PROGRAM MAIN
VAR
	onTimer, offTimer : ton;
	
	start : BOOL;
END_VAR

onTimer(PT:=T#1S, Q=> GVL.imAlive);
offTimer(IN:= GVl.imAlive, PT:=T#1S);
IF offTimer.Q THEN
	onTimer.IN := FALSE;
END_IF
IF NOT GVL.imAlive AND NOT onTimer.IN THEN
	onTimer.IN := TRUE;
	GVL.counter := GVL.counter +1;
END_IF

END_PROGRAM

(* stored: Version 1.1.0.1, ProductVersion 3.1.4024.3
   POU MAIN: Id {3e163404-f789-4a48-8427-1d9c1477f42e}, SpecialFunc None *)
